FUNCTION_BLOCK FB_OilPump
VAR_INPUT
	i_bCallForCyl: BOOL := TRUE;
END_VAR
VAR_OUTPUT
END_VAR
VAR
    iState : INT := 0;
	FeedbackTimer : TON;
    DelayTimer : TON;
END_VAR

CASE iState OF
    0: (* Pump Off, Not Enabled *)
        iState := 10;

    10: (* Pump Enabled from Other Routine *)
		IF GVL_IO.DI_M1 THEN
			DelayAndAdvance( GVL_InitialSetting.PUMP_FAN_DelayTime, iState+1 );
		END_IF
	11:
		GVL_IO.DO_M2 := TRUE;
	    (* Inhibit Pump if DI1.4 or DI1.5 goes Low *)
        IF (NOT GVL_IO.DI_LS1) OR (NOT GVL_IO.DI_TS1) THEN
			GVL_IO.DO_M1 := FALSE;
			GVL_IO.DO_M2 := FALSE;
            iState := iState + 1;
        END_IF
	12: // check to off pump
		IF NOT GVL_IO.DI_M1 THEN
			FB_CheckFeedback( t := E_FT.PUMP, FeedbackTimer := FeedbackTimer );
		ELSE
			iState := (iState + 10) / 10 * 10;
        END_IF

    20: (* Fault Handling: Check DI1.3 Feedback *)
        (* Start 3-second timer to check for DI1.3 feedback *)
        DelayAndAdvance( GVL_InitialSetting.PUMP_RestartingTime, iState+1 );
	21:
        IF NOT GVL_IO.DI_M1 THEN
			GVL_HMI.i_nPumpState := -1;
			FB_SetAlarm( sMsg:=GVL_AlarmMessage.PUMP );
			iState := iState / 10 * 10;
		ELSE
			iState := (iState + 10) / 10 * 10;
        END_IF
END_CASE

METHOD DelayAndAdvance : BOOL
VAR_INPUT
	i_nDelayTime: INT;	// ms
	i_nNextState: INT;
END_VAR

VAR
END_VAR
IF NOT DelayTimer.IN THEN
    DelayTimer(IN := TRUE, PT := INT_TO_TIME(i_nDelayTime));
ELSE
    IF DelayTimer.Q THEN 
        iState := i_nNextState; 
    END_IF
END_IF
END_METHOD

END_FUNCTION_BLOCK

(* stored: Version 1.1.0.1, ProductVersion 3.1.4024.6
   POU FB_OilPump: Id {eb1edbee-9a4b-4f1e-8695-a5d69ca2499b}, SpecialFunc None
   Method DelayAndAdvance: Id {c0f40f36-8a2d-4f35-96c3-ddd282aa94ff} *)
